# EPICS autosave request: ip/ipApp/Db/picoMotor_positions.req
# FILE... picoMotor_positions.req
$(P)$(S):$(D):pM$(M)_pos.VAL
$(P)$(S):$(D):pM$(M)_prev.VAL
